INTERFACE ITF_Group1_HMI_Connector_View EXTENDS ITF_BaseGroupElement_HMI_Connector_View

END_INTERFACE

(* stored: Version 1.1.0.1
   Itf ITF_Group1_HMI_Connector_View: Id {9ffe63b4-d4e1-01ec-3745-4b6b555b6a66} *)
